FUNCTION HLI_ChannelModeAuto : BOOL
VAR_INPUT
	nChan					: UDINT;			(* Number of channel *)
	ProgramName 		: STRING(HLI_IMCM_MODE_STATE_PARAM_STRL);
	pUnit					: POINTER TO MC_CONTROL_MCM_MODE_STATE_UNIT;
	pCommand				: POINTER TO HLI_PROC_TRANS_TO_MODE_STATE;
	pChannel				: POINTER TO ST_CncChannel;
END_VAR
VAR
	pString				: POINTER TO STRING(HLI_IMCM_MODE_STATE_PARAM_STRL);
END_VAR

(* ========================================================= *)
(*    FUN: HLI_ChannelModeAuto                               *)
(* --------------------------------------------------------- *)
(*   Desc: switch channel to Automatic mode / xxx            *)
(* Author: MK                                                *)
(*   Date: 18.07.2002                                        *)
(*   Rev.: 1.0                                               *)
(* ========================================================= *)


IF pChannel^.State.Selected THEN
	pChannel^.State.Selected := FALSE;
	pCommand^.to_mode := HLI_IMCM_AUTOMATIC_MODE;
	pCommand^.to_state := HLI_IMCM_PROCESS_SELECTED;
	pCommand^.channel_number := nChan;
	pString := ADR(pCommand^.parameter);
	pString^ := ProgramName;
	pUnit^.command_semaphor_rw := TRUE;
	ADSLOG(strMsg:='Automatic selected', nDINT:=0, strArg := '');
END_IF

 
IF GVL.gvl_automaticselected THEN
	pChannel^.State.Selected := FALSE;
	pCommand^.to_mode := HLI_IMCM_AUTOMATIC_MODE;
	pCommand^.to_state := HLI_IMCM_PROCESS_SELECTED;
	pCommand^.channel_number := nChan;
	pString := ADR(pCommand^.parameter);
	pString^ := ProgramName;
	pUnit^.command_semaphor_rw := TRUE;
	ADSLOG(strMsg:='Automatic selected', nDINT:=0, strArg := '');
END_IF


IF pChannel^.State.Ready THEN
	pChannel^.State.Ready := FALSE;
	pCommand^.to_mode := HLI_IMCM_AUTOMATIC_MODE;
	pCommand^.to_state := HLI_IMCM_PROCESS_READY;
	pCommand^.channel_number := nChan;
	pString := ADR(pCommand^.parameter);
	pString^ := ProgramName;
	pUnit^.command_semaphor_rw := TRUE;
	ADSLOG(strMsg:='Automatic ready', nDINT:=0, strArg := '');
END_IF

IF pChannel^.State.Start THEN
	pChannel^.State.Start := FALSE;
	pCommand^.to_mode := HLI_IMCM_AUTOMATIC_MODE;
	pCommand^.to_state := HLI_IMCM_PROCESS_ACTIVE;
	pCommand^.channel_number := nChan;
	pString := ADR(pCommand^.parameter);
	pString^ := ProgramName;
	pUnit^.command_semaphor_rw := TRUE;
	ADSLOG(strMsg:='Programm %s started', nDINT:=0, strArg:=ProgramName);
END_IF

 //IF pChannel^.State.Stop THEN
IF GVL.gvl_automaticstop THEN
	pChannel^.State.Stop := FALSE;
	pCommand^.to_mode := HLI_IMCM_AUTOMATIC_MODE;
	pCommand^.to_state := HLI_IMCM_PROCESS_HOLD;
	pCommand^.channel_number := nChan;
	pUnit^.command_semaphor_rw := TRUE;
	ADSLOG(strMsg:='Programm stopped', nDINT:=0, strArg := '');
END_IF

//IF pChannel^.State.Reset THEN
IF GVL.gvl_automaticreset THEN
	pChannel^.State.Reset := FALSE;
	pCommand^.to_mode := HLI_IMCM_AUTOMATIC_MODE;
	pCommand^.to_state := HLI_IMCM_PROCESS_DESELECTED;
	pCommand^.channel_number := nChan;
	pUnit^.command_semaphor_rw := TRUE;
	ADSLOG(strMsg:='Automatic resetting', nDINT:=0, strArg := '');
END_IF

HLI_ChannelModeAuto := TRUE;

END_FUNCTION

(* stored: Version 1.1.0.1, ProductVersion 3.1.4020.12
   POU HLI_ChannelModeAuto: Id {3e9182a1-775e-4f58-aa4a-e0eef786107f}, SpecialFunc None *)
